TYPE UNIFIED_PROGRAM_STEP_TRANSITION_CONDITION :
STRUCT
	Name : STRING;
	Args : ARRAY [0..UnifiedProgramConstants.MaxActionArgumentsCount - 1] OF STRING(255);
END_STRUCT
END_TYPE

(* stored: Version 1.1.0.1
   DUT UNIFIED_PROGRAM_STEP_TRANSITION_CONDITION: Id {4ffbbe1b-92b6-4911-a124-aa6ba709d0a6} *)
